// TwinCAT 3 PLC project LibraryVision
// Title: LibraryVision
// Company: Gema
// Author: RG
// ProjectVersion: 0.9.9.9
// ProgramVersion: 3.1.4024.0
// libraries:
//   Tc2_EtherCAT, * (Beckhoff Automation GmbH)
//   Tc2_System, * (Beckhoff Automation GmbH)
//   TcoCore, 0.11.0.23 (Vortex.Library)
//   TcoData, 0.11.0.23 (Vortex.Library)
//   TcoDrivesBeckhoff, 0.11.0.23 (Vortex.Library)
//   TcoElements, 0.11.0.23 (Vortex.Library)
//   TcoIo, 0.11.0.23 (Vortex.Library)
//   TcoPneumatics, 0.11.0.23 (Vortex.Library)
// project tree:
//   Context/ MainStation.TcPOU, PRG_TEST.TcPOU, TcUnitContext.TcPOU
//   IV3/Dut/CoE/ GeneralDeviceInformation.TcDUT, IdentityCoe.TcDUT
//   IV3/Dut/ Coordinates.TcDUT, FieldOfView.TcDUT
//   IV3/Dut/IO/Base/ EtcMasterBase_62654B43.TcDUT, EtcSlaveBase_82538BE2.TcDUT, EtcSlaveBoxBase_77A0E4A7.TcDUT, EtcSlaveEndTerminalBase_866C7F0C.TcDUT, EtcSlaveTerminalBase_947E5A46.TcDUT, InputBase_8311D824.TcDUT, OutputBase_10CEE7DE.TcDUT, SyncUnitsBase_AD6C35CE.TcDUT, SyncUnitTaskBase_FCD3CBF3.TcDUT, SyncUnitTasksBase_7C8711EB.TcDUT
//   IV3/Dut/IO/Devices/ SyncUnits_67D36DDA.TcDUT, SyncUnitTasks_4BE01469.TcDUT, SyncUnitTask_AB2F5079.TcDUT
//   IV3/Dut/IO/PDOs/BitValues/ Iv3InputRequestResponse1.TcDUT, Iv3InputRequestResponse2.TcDUT, Iv3InputRequestResponse3.TcDUT, Iv3InputRequestResponse4.TcDUT (not stored), Iv3InputRequestResponse5.TcDUT
//   IV3/Dut/IO/PDOs/ ID01_Current_Value.TcDUT, ID01_Status.TcDUT, ID02_Current_Value.TcDUT, ID02_Status.TcDUT, ID03_Current_Value.TcDUT, ID03_Status.TcDUT, ID04_Current_Value.TcDUT, ID04_Status.TcDUT, ID05_Current_Value.TcDUT, ID05_Status.TcDUT, ID06_Current_Value.TcDUT, ID06_Status.TcDUT, ID07_Current_Value.TcDUT, ID07_Status.TcDUT, ID08_Current_Value.TcDUT, ID08_Status.TcDUT, InfoData.TcDUT, InfoData_8649EEEB.TcDUT, InfoData_E68C61CD.TcDUT, Inputs.TcDUT, Input_Request.TcDUT, Input_Response.TcDUT, Outputs.TcDUT, Status_of_System.TcDUT, WcState_0B2B16F9.TcDUT, WcState_9091E0EB.TcDUT
//   IV3/Interfaces/ iCalculationTask.TcIO
//   IV3/ IVController.TcPOU
//   IV3/Tasks/ ReadCoordinates.TcPOU, CalculationTask.TcPOU, TriggerSensor.TcPOU
//   Project Information/ F_GetCompany.TcPOU, F_GetTitle.TcPOU, F_GetVersion.TcPOU
//   Version/ Global_Version.TcGVL
// real-time tasks:
//   TASK PlcTask: cycle T#1ms, priority 20, ADS port 350
// I/O:
//   DEVICE Device 2 (EtherCAT), AmsNetId 192.168.1.8.3.1
//     IV3_Sensor1(DL-EC1A)
// variable links:
//   LibraryVisionExample Instance <-> Device 2 (EtherCAT)/IV3_Sensor1(DL-EC1A)
//     PlcTask Inputs/MAIN._app._mainStation._IvController.ID01Status/Change_Program_Ack <-> ID01 Status/Change Program Ack
//     PlcTask Inputs/MAIN._app._mainStation._IvController.ID01Status/Change_Program_Failed <-> ID01 Status/Change Program Failed
//     PlcTask Inputs/MAIN._app._mainStation._IvController.ID01Status/Error_status <-> ID01 Status/Error status
//     PlcTask Inputs/MAIN._app._mainStation._IvController.ID01Status/Program_Num_00 <-> ID01 Status/Program Num 00
//     PlcTask Inputs/MAIN._app._mainStation._IvController.ID02Status/Program_Num_01 <-> ID02 Status/Program Num 01
//     PlcTask Inputs/MAIN._app._mainStation._IvController.ID03Status/Program_Num_02 <-> ID03 Status/Program Num 02
//     PlcTask Inputs/MAIN._app._mainStation._IvController.ID04Status/Program_Num_03 <-> ID04 Status/Program Num 03
//     PlcTask Inputs/MAIN._app._mainStation._IvController.ID05Status/Program_Num_04 <-> ID05 Status/Program Num 04
//     PlcTask Inputs/MAIN._app._mainStation._IvController.ID06Status/Program_Num_05 <-> ID06 Status/Program Num 05
//     PlcTask Inputs/MAIN._app._mainStation._IvController.ID07Status/Program_Num_06 <-> ID07 Status/Program Num 06
//     PlcTask Inputs/MAIN._app._mainStation._IvController.ID01Status/Result_Valid <-> ID01 Status/Result Valid
//     PlcTask Inputs/MAIN._app._mainStation._IvController.ID01Status/Total_Status_OK <-> ID01 Status/Total Status OK
//     PlcTask Inputs/MAIN._app._mainStation._IvController.ID03Status/Total_Status_OK <-> ID03 Status/Total Status OK
//     PlcTask Inputs/MAIN._app._mainStation._IvController.ID01_CurrentValue/Reserved <-> ID01 Current Value/Reserved
//     PlcTask Inputs/MAIN._app._mainStation._IvController.ID02Status/Result_Updated_Toggle <-> ID02 Status/Result Updated Toggle
//     PlcTask Inputs/MAIN._app._mainStation._IvController.ID02Status/Tool_00_Invalid <-> ID02 Status/Tool 00 Invalid
//     PlcTask Inputs/MAIN._app._mainStation._IvController.ID03Status/Tool_01_Invalid <-> ID03 Status/Tool 01 Invalid
//     PlcTask Inputs/MAIN._app._mainStation._IvController.ID04Status/Tool_02_Invalid <-> ID04 Status/Tool 02 Invalid
//     PlcTask Inputs/MAIN._app._mainStation._IvController.ID05Status/Tool_03_Invalid <-> ID05 Status/Tool 03 Invalid
//     PlcTask Inputs/MAIN._app._mainStation._IvController.ID06Status/Tool_04_Invalid <-> ID06 Status/Tool 04 Invalid
//     PlcTask Inputs/MAIN._app._mainStation._IvController.ID07Status/Tool_05_Invalid <-> ID07 Status/Tool 05 Invalid
//     PlcTask Inputs/MAIN._app._mainStation._IvController.ID08Status/Tool_06_Invalid <-> ID08 Status/Tool 06 Invalid
//     PlcTask Inputs/MAIN._app._mainStation._IvController.ID02Status/Tool_00_Status <-> ID02 Status/Tool 00 Status
//     PlcTask Inputs/MAIN._app._mainStation._IvController.ID03Status/Tool_01_Status <-> ID03 Status/Tool 01 Status
//     PlcTask Inputs/MAIN._app._mainStation._IvController.ID04Status/Tool_02_Status <-> ID04 Status/Tool 02 Status
//     PlcTask Inputs/MAIN._app._mainStation._IvController.ID05Status/Tool_03_Status <-> ID05 Status/Tool 03 Status
//     PlcTask Inputs/MAIN._app._mainStation._IvController.ID06Status/Tool_04_Status <-> ID06 Status/Tool 04 Status
//     PlcTask Inputs/MAIN._app._mainStation._IvController.ID07Status/Tool_05_Status <-> ID07 Status/Tool 05 Status
//     PlcTask Inputs/MAIN._app._mainStation._IvController.ID08Status/Tool_06_Status <-> ID08 Status/Tool 06 Status
//     PlcTask Inputs/MAIN._app._mainStation._IvController.ID02Status/Trigger_Ack <-> ID02 Status/Trigger Ack
//     PlcTask Inputs/MAIN._app._mainStation._IvController.ID02Status/Trigger_Failed <-> ID02 Status/Trigger Failed
//     PlcTask Inputs/MAIN._app._mainStation._IvController.ID02_MatchingRateOfPositionAdujustmentTool_01/Tool_00_Score <-> ID02 Current Value/Tool 00 Score
//     PlcTask Inputs/MAIN._app._mainStation._IvController.ID03_MatchingRateOfPositionAdujustmentTool_02/Tool_01_Score <-> ID03 Current Value/Tool 01 Score
//     PlcTask Inputs/MAIN._app._mainStation._IvController.ID04_MatchingRateOfPositionAdujustmentTool_03/Tool_02_Score <-> ID04 Current Value/Tool 02 Score
//     PlcTask Inputs/MAIN._app._mainStation._IvController.ID05_MatchingRateOfPositionAdujustmentTool_04/Tool_03_Score <-> ID05 Current Value/Tool 03 Score
//     PlcTask Inputs/MAIN._app._mainStation._IvController.ID06_MatchingRateOfPositionAdujustmentTool_05/Tool_04_Score <-> ID06 Current Value/Tool 04 Score
//     PlcTask Inputs/MAIN._app._mainStation._IvController.ID07_MatchingRateOfPositionAdujustmentTool_06/Tool_05_Score <-> ID07 Current Value/Tool 05 Score
//     PlcTask Inputs/MAIN._app._mainStation._IvController.ID08_MatchingRateOfPositionAdujustmentTool_07/Tool_06_Score <-> ID08 Current Value/Tool 06 Score
//     PlcTask Inputs/MAIN._app._mainStation._IvController.ID03Status/Regist_Master_Image_Ack <-> ID03 Status/Regist Master Image Ack
//     PlcTask Inputs/MAIN._app._mainStation._IvController.ID03Status/Regist_Master_Image_Failed <-> ID03 Status/Regist Master Image Failed
//     PlcTask Inputs/MAIN._app._mainStation._IvController.ID04Status/Logic_01 <-> ID04 Status/Logic 01
//     PlcTask Inputs/MAIN._app._mainStation._IvController.ID05Status/Logic_02 <-> ID05 Status/Logic 02
//     PlcTask Inputs/MAIN._app._mainStation._IvController.ID06Status/Logic_03 <-> ID06 Status/Logic 03
//     PlcTask Inputs/MAIN._app._mainStation._IvController.ID07Status/Logic_04 <-> ID07 Status/Logic 04
//     PlcTask Inputs/MAIN._app._mainStation._IvController.ID04Status/SD_Card_Detected <-> ID04 Status/SD Card Detected
//     PlcTask Inputs/MAIN._app._mainStation._IvController.ID04Status/SD_Save_Stop_Ack <-> ID04 Status/SD Save Stop Ack
//     PlcTask Inputs/MAIN._app._mainStation._IvController.ID05Status/Reset_Statistics_Ack <-> ID05 Status/Reset Statistics Ack
//     PlcTask Inputs/MAIN._app._mainStation._IvController.ID05Status/Run <-> ID05 Status/Run
//     PlcTask Inputs/MAIN._app._mainStation._IvController.ID06Status/Busy <-> ID06 Status/Busy
//     PlcTask Inputs/MAIN._app._mainStation._IvController.ID06Status/Clear_Error_Ack <-> ID06 Status/Clear Error Ack
//     PlcTask Inputs/MAIN._app._mainStation._IvController.ID08Status/SD_Card_No_Space <-> ID08 Status/SD Card No Space
//     PlcTask Inputs/MAIN._app._mainStation._IvController.ID08Status/Total_Status_NG <-> ID08 Status/Total Status NG
//     PlcTask Inputs/MAIN._app._mainStation._IvController.InfoData/AdsAddr <-> InfoData/AdsAddr
//     PlcTask Inputs/MAIN._app._mainStation._IvController.InfoData/State <-> InfoData/State
//     PlcTask Inputs/MAIN._app._mainStation._IvController.InputResponse/Response_{1..5} <-> Input Response {1..5}/Reserved  (5 links)
//     PlcTask Inputs/MAIN._app._mainStation._IvController.StatusOfSystem/Error_Code <-> Status of System/Error Code
//     PlcTask Inputs/MAIN._app._mainStation._IvController.StatusOfSystem/Error_Status <-> Status of System/Error Status
//     PlcTask Inputs/MAIN._app._mainStation._IvController.WcState/WcState <-> WcState/WcState
//     PlcTask Outputs/MAIN._app._mainStation._IvController.InputRequest/Request_{1..5} <-> Input Request {1..5}/Request {1..5}  (5 links)

// ---- IV3/Dut/CoE/GeneralDeviceInformation.TcDUT
TYPE
    GeneralDeviceInformation :
    STRUCT
        DeviceType      : UDINT;
        DeviceName      : STRING;
        HardwareVersion : STRING;
        SoftwareVersion : STRING;
    END_STRUCT
END_TYPE

// ---- IV3/Dut/CoE/IdentityCoe.TcDUT
TYPE
    IdentityCoe :
    STRUCT
        VendorId     : DWORD;
        ProductKey   : DWORD;
        Revision     : DWORD;
        SerialNumber : DWORD;
    END_STRUCT
END_TYPE

// ---- IV3/Dut/Coordinates.TcDUT
TYPE
    Coordinates :
    STRUCT
        xValue        : DINT;
        yValue        : DINT;
        variableValue : DINT;
    END_STRUCT
END_TYPE

// ---- IV3/Dut/FieldOfView.TcDUT
TYPE
    FieldOfView :
    STRUCT
        xValue : LREAL;
        yValue : lreal;
    END_STRUCT
END_TYPE

// ---- IV3/Dut/IO/Base/EtcMasterBase_62654B43.TcDUT

TYPE
    EtcMasterBase_62654B43 :
    STRUCT
    END_STRUCT
END_TYPE

// ---- IV3/Dut/IO/Base/EtcSlaveBase_82538BE2.TcDUT

TYPE
    EtcSlaveBase_82538BE2 :
    STRUCT
    END_STRUCT
END_TYPE

// ---- IV3/Dut/IO/Base/EtcSlaveBoxBase_77A0E4A7.TcDUT

{attribute clr[Container(Layout.Stack)]}
{attribute clr[Group(Layout.GroupBox)]}
{attribute addProperty PreviousPort "Unknown"}
{attribute addProperty SyncUnit "Unknown"}
TYPE
    EtcSlaveBoxBase_77A0E4A7 EXTENDS EtcSlaveBase_82538BE2 :
    STRUCT
    END_STRUCT
END_TYPE

// ---- IV3/Dut/IO/Base/EtcSlaveEndTerminalBase_866C7F0C.TcDUT

{attribute clr[Container(Layout.Stack)]}
{attribute clr[Group(Layout.GroupBox)]}
{attribute addProperty PreviousPort "Unknown"}
{attribute addProperty SyncUnit "Unknown"}
TYPE
    EtcSlaveEndTerminalBase_866C7F0C EXTENDS EtcSlaveBase_82538BE2 :
    STRUCT
    END_STRUCT
END_TYPE

// ---- IV3/Dut/IO/Base/EtcSlaveTerminalBase_947E5A46.TcDUT

{attribute clr[Container(Layout.Stack)]}
{attribute clr[Group(Layout.GroupBox)]}
{attribute addProperty PreviousPort "Unknown"}
{attribute addProperty SyncUnit "Unknown"}
TYPE
    EtcSlaveTerminalBase_947E5A46 EXTENDS EtcSlaveBase_82538BE2 :
    STRUCT
    END_STRUCT
END_TYPE

// ---- IV3/Dut/IO/Base/InputBase_8311D824.TcDUT

TYPE
    InputBase_8311D824 :
    STRUCT
    END_STRUCT
END_TYPE

// ---- IV3/Dut/IO/Base/OutputBase_10CEE7DE.TcDUT

TYPE
    OutputBase_10CEE7DE :
    STRUCT
    END_STRUCT
END_TYPE

// ---- IV3/Dut/IO/Base/SyncUnitsBase_AD6C35CE.TcDUT

TYPE
    SyncUnitsBase_AD6C35CE :
    STRUCT
    END_STRUCT
END_TYPE

// ---- IV3/Dut/IO/Base/SyncUnitTaskBase_FCD3CBF3.TcDUT

TYPE
    SyncUnitTaskBase_FCD3CBF3 :
    STRUCT
    END_STRUCT
END_TYPE

// ---- IV3/Dut/IO/Base/SyncUnitTasksBase_7C8711EB.TcDUT

TYPE
    SyncUnitTasksBase_7C8711EB :
    STRUCT
    END_STRUCT
END_TYPE

// ---- IV3/Dut/IO/Devices/SyncUnits_67D36DDA.TcDUT
{attribute 'GeneratedUsingTerminal: '}
{attribute addProperty BoxType ""}
{attribute addProperty Id "_defaultAT %I*SyncUnitTasks_4BE0146918"}
{attribute addProperty CRC "1741909466"}
{attribute addProperty Size "18"}
TYPE
    SyncUnits_67D36DDA EXTENDS SyncUnitsBase_AD6C35CE :
    STRUCT
        {attribute addProperty Name "_default"}
        _default : SyncUnitTasks_4BE01469;
    END_STRUCT
END_TYPE

// ---- IV3/Dut/IO/Devices/SyncUnitTasks_4BE01469.TcDUT
{attribute 'GeneratedUsingTerminal: '}
{attribute addProperty BoxType ""}
{attribute addProperty Id "unreferencedAT %I*SyncUnitTask_AB2F50799PlcTaskAT %I*SyncUnitTask_AB2F50799"}
{attribute addProperty CRC "1272976489"}
{attribute addProperty Size "18"}
TYPE
    SyncUnitTasks_4BE01469 EXTENDS SyncUnitTasksBase_7C8711EB :
    STRUCT
        {attribute addProperty Name "unreferenced"}
        unreferenced : SyncUnitTask_AB2F5079;
        {attribute addProperty Name "PlcTask"}
        PlcTask : SyncUnitTask_AB2F5079;
    END_STRUCT
END_TYPE

// ---- IV3/Dut/IO/Devices/SyncUnitTask_AB2F5079.TcDUT
{attribute 'GeneratedUsingTerminal: IODEVICETYPE_ETHERCATPROT'}
{attribute addProperty BoxType "IODEVICETYPE_ETHERCATPROT"}
{attribute addProperty Id "WcStateAT %I*WcState_0B2B16F91InfoDataAT %I*InfoData_8649EEEB8"}
{attribute addProperty CRC "2872004729"}
{attribute addProperty Size "9"}
TYPE
    SyncUnitTask_AB2F5079 EXTENDS SyncUnitTaskBase_FCD3CBF3 :
    STRUCT
        {attribute addProperty Name "WcState"}
        WcState : WcState_0B2B16F9;
        {attribute addProperty Name "InfoData"}
        InfoData : InfoData_8649EEEB;
    END_STRUCT
END_TYPE

// ---- IV3/Dut/IO/PDOs/BitValues/Iv3InputRequestResponse1.TcDUT
//Index0x7000   Subindex 16#1
TYPE
    Iv3InputRequestResponse1 :
    STRUCT
        Bit0                      : BIT;
        ProgramChangeRequest      : BIT;
        Trigger                   : BIT;
        MasterRegistrationRequest : BIT;
        MemoryStopSdCardRequest   : BIT;
        ResetStatistics           : BIT;
        ResetError                : BIT;
        Bit7                      : BIT;
        Bit8                      : BIT;
        Bit9                      : BIT;
        Bit10                     : BIT;
        Bit11                     : BIT;
        Bit12                     : BIT;
        Bit13                     : BIT;
        Bit14                     : BIT;
        Bit15                     : BIT;

    END_STRUCT
END_TYPE

// ---- IV3/Dut/IO/PDOs/BitValues/Iv3InputRequestResponse2.TcDUT
//Index0x7000   Subindex 16#2
TYPE
    Iv3InputRequestResponse2 :
    STRUCT
        Bit0                     : BIT;
        SwitchProgrammNumberBit0 : BIT;
        Bit2                     : BIT;
        Bit3                     : BIT;
        Bit4                     : BIT;
        Bit5                     : BIT;
        Bit6                     : BIT;
        Bit7                     : BIT;
        Bit8                     : BIT;
        Bit9                     : BIT;
        Bit10                    : BIT;
        Bit11                    : BIT;
        Bit12                    : BIT;
        Bit13                    : BIT;
        Bit14                    : BIT;
        Bit15                    : BIT;

    END_STRUCT
END_TYPE

// ---- IV3/Dut/IO/PDOs/BitValues/Iv3InputRequestResponse3.TcDUT
//Index0x7000   Subindex 16#3
TYPE
    Iv3InputRequestResponse3 :
    STRUCT
        Bit0                     : BIT;
        SwitchProgrammNumberBit1 : BIT;
        Bit2                     : BIT;
        Bit3                     : BIT;
        Bit4                     : BIT;
        Bit5                     : BIT;
        Bit6                     : BIT;
        Bit7                     : BIT;
        Bit8                     : BIT;
        Bit9                     : BIT;
        Bit10                    : BIT;
        Bit11                    : BIT;
        Bit12                    : BIT;
        Bit13                    : BIT;
        Bit14                    : BIT;
        Bit15                    : BIT;

    END_STRUCT
END_TYPE

// ---- IV3/Dut/IO/PDOs/BitValues/Iv3InputRequestResponse5.TcDUT
//Index0x7000   Subindex 16#5
TYPE
    Iv3InputRequestResponse5 :
    STRUCT
        Bit0                     : BIT;
        SwitchProgrammNumberBit3 : BIT;
        Bit2                     : BIT;
        Bit3                     : BIT;
        Bit4                     : BIT;
        Bit5                     : BIT;
        Bit6                     : BIT;
        Bit7                     : BIT;
        Bit8                     : BIT;
        Bit9                     : BIT;
        Bit10                    : BIT;
        Bit11                    : BIT;
        Bit12                    : BIT;
        Bit13                    : BIT;
        Bit14                    : BIT;
        Bit15                    : BIT;

    END_STRUCT
END_TYPE

// ---- IV3/Dut/IO/PDOs/ID01_Current_Value.TcDUT
{attribute 'GeneratedUsingTerminal: DL-EC1A-0000'}
{attribute addProperty BoxType "DL-EC1A-0000"}
{attribute addProperty Id "ReservedAT %I*DINT4"}
{attribute addProperty CRC "2013026300"}
{attribute addProperty Size "4"}
TYPE
    ID01_Current_Value EXTENDS InputBase_8311D824 :
    STRUCT
        {attribute addProperty Name "Reserved"}
        Reserved AT %I* : DINT;
    END_STRUCT
END_TYPE

// ---- IV3/Dut/IO/PDOs/ID01_Status.TcDUT
{attribute 'GeneratedUsingTerminal: DL-EC1A-0000'}
{attribute addProperty BoxType "DL-EC1A-0000"}
{attribute addProperty Id "Change_Program_AckAT %I*BOOL1Change_Program_FailedAT %I*BOOL1Result_ValidAT %I*BOOL1Total_Status_OKAT %I*BOOL1Program_Num_00AT %I*BOOL1Error_statusAT %I*BOOL1"}
{attribute addProperty CRC "3787914147"}
{attribute addProperty Size "6"}
TYPE
    ID01_Status EXTENDS InputBase_8311D824 :
    STRUCT
        {attribute addProperty Name "Change_Program_Ack"}
        Change_Program_Ack AT %I* : BOOL;
        {attribute addProperty Name "Change_Program_Failed"}
        Change_Program_Failed AT %I* : BOOL;
        {attribute addProperty Name "Result_Valid"}
        Result_Valid AT %I* : BOOL;
        {attribute addProperty Name "Total_Status_OK"}
        Total_Status_OK AT %I* : BOOL;
        {attribute addProperty Name "Program_Num_00"}
        Program_Num_00 AT %I* : BOOL;
        {attribute addProperty Name "Error_status"}
        Error_status AT %I* : BOOL;
    END_STRUCT
END_TYPE

// ---- IV3/Dut/IO/PDOs/ID02_Current_Value.TcDUT
{attribute 'GeneratedUsingTerminal: DL-EC1A-0000'}
{attribute addProperty BoxType "DL-EC1A-0000"}
{attribute addProperty Id "Tool_00_ScoreAT %I*DINT4"}
{attribute addProperty CRC "539608926"}
{attribute addProperty Size "4"}
TYPE
    ID02_Current_Value EXTENDS InputBase_8311D824 :
    STRUCT
        {attribute addProperty Name "Tool_00_Score"}
        Tool_00_Score AT %I* : DINT;
    END_STRUCT
END_TYPE

// ---- IV3/Dut/IO/PDOs/ID02_Status.TcDUT
{attribute 'GeneratedUsingTerminal: DL-EC1A-0000'}
{attribute addProperty BoxType "DL-EC1A-0000"}
{attribute addProperty Id "Trigger_AckAT %I*BOOL1Trigger_FailedAT %I*BOOL1Result_Updated_ToggleAT %I*BOOL1Tool_00_StatusAT %I*BOOL1Program_Num_01AT %I*BOOL1Tool_00_InvalidAT %I*BOOL1"}
{attribute addProperty CRC "3351424392"}
{attribute addProperty Size "6"}
TYPE
    ID02_Status EXTENDS InputBase_8311D824 :
    STRUCT
        {attribute addProperty Name "Trigger_Ack"}
        Trigger_Ack AT %I* : BOOL;
        {attribute addProperty Name "Trigger_Failed"}
        Trigger_Failed AT %I* : BOOL;
        {attribute addProperty Name "Result_Updated_Toggle"}
        Result_Updated_Toggle AT %I* : BOOL;
        {attribute addProperty Name "Tool_00_Status"}
        Tool_00_Status AT %I* : BOOL;
        {attribute addProperty Name "Program_Num_01"}
        Program_Num_01 AT %I* : BOOL;
        {attribute addProperty Name "Tool_00_Invalid"}
        Tool_00_Invalid AT %I* : BOOL;
    END_STRUCT
END_TYPE

// ---- IV3/Dut/IO/PDOs/ID03_Current_Value.TcDUT
{attribute 'GeneratedUsingTerminal: DL-EC1A-0000'}
{attribute addProperty BoxType "DL-EC1A-0000"}
{attribute addProperty Id "Tool_01_ScoreAT %I*DINT4"}
{attribute addProperty CRC "2706247979"}
{attribute addProperty Size "4"}
TYPE
    ID03_Current_Value EXTENDS InputBase_8311D824 :
    STRUCT
        {attribute addProperty Name "Tool_01_Score"}
        Tool_01_Score AT %I* : DINT;
    END_STRUCT
END_TYPE

// ---- IV3/Dut/IO/PDOs/ID03_Status.TcDUT
{attribute 'GeneratedUsingTerminal: DL-EC1A-0000'}
{attribute addProperty BoxType "DL-EC1A-0000"}
{attribute addProperty Id "Regist_Master_Image_AckAT %I*BOOL1Regist_Master_Image_FailedAT %I*BOOL1Total_Status_OKAT %I*BOOL1Tool_01_StatusAT %I*BOOL1Program_Num_02AT %I*BOOL1Tool_01_InvalidAT %I*BOOL1"}
{attribute addProperty CRC "695297954"}
{attribute addProperty Size "6"}
TYPE
    ID03_Status EXTENDS InputBase_8311D824 :
    STRUCT
        {attribute addProperty Name "Regist_Master_Image_Ack"}
        Regist_Master_Image_Ack AT %I* : BOOL;
        {attribute addProperty Name "Regist_Master_Image_Failed"}
        Regist_Master_Image_Failed AT %I* : BOOL;
        {attribute addProperty Name "Total_Status_OK"}
        Total_Status_OK AT %I* : BOOL;
        {attribute addProperty Name "Tool_01_Status"}
        Tool_01_Status AT %I* : BOOL;
        {attribute addProperty Name "Program_Num_02"}
        Program_Num_02 AT %I* : BOOL;
        {attribute addProperty Name "Tool_01_Invalid"}
        Tool_01_Invalid AT %I* : BOOL;
    END_STRUCT
END_TYPE

// ---- IV3/Dut/IO/PDOs/ID04_Current_Value.TcDUT
{attribute 'GeneratedUsingTerminal: DL-EC1A-0000'}
{attribute addProperty BoxType "DL-EC1A-0000"}
{attribute addProperty Id "Tool_02_ScoreAT %I*DINT4"}
{attribute addProperty CRC "640120323"}
{attribute addProperty Size "4"}
TYPE
    ID04_Current_Value EXTENDS InputBase_8311D824 :
    STRUCT
        {attribute addProperty Name "Tool_02_Score"}
        Tool_02_Score AT %I* : DINT;
    END_STRUCT
END_TYPE

// ---- IV3/Dut/IO/PDOs/ID04_Status.TcDUT
{attribute 'GeneratedUsingTerminal: DL-EC1A-0000'}
{attribute addProperty BoxType "DL-EC1A-0000"}
{attribute addProperty Id "SD_Save_Stop_AckAT %I*BOOL1SD_Card_DetectedAT %I*BOOL1Logic_01AT %I*BOOL1Tool_02_StatusAT %I*BOOL1Program_Num_03AT %I*BOOL1Tool_02_InvalidAT %I*BOOL1"}
{attribute addProperty CRC "922163961"}
{attribute addProperty Size "6"}
TYPE
    ID04_Status EXTENDS InputBase_8311D824 :
    STRUCT
        {attribute addProperty Name "SD_Save_Stop_Ack"}
        SD_Save_Stop_Ack AT %I* : BOOL;
        {attribute addProperty Name "SD_Card_Detected"}
        SD_Card_Detected AT %I* : BOOL;
        {attribute addProperty Name "Logic_01"}
        Logic_01 AT %I* : BOOL;
        {attribute addProperty Name "Tool_02_Status"}
        Tool_02_Status AT %I* : BOOL;
        {attribute addProperty Name "Program_Num_03"}
        Program_Num_03 AT %I* : BOOL;
        {attribute addProperty Name "Tool_02_Invalid"}
        Tool_02_Invalid AT %I* : BOOL;
    END_STRUCT
END_TYPE

// ---- IV3/Dut/IO/PDOs/ID05_Current_Value.TcDUT
{attribute 'GeneratedUsingTerminal: DL-EC1A-0000'}
{attribute addProperty BoxType "DL-EC1A-0000"}
{attribute addProperty Id "Tool_03_ScoreAT %I*DINT4"}
{attribute addProperty CRC "2806030454"}
{attribute addProperty Size "4"}
TYPE
    ID05_Current_Value EXTENDS InputBase_8311D824 :
    STRUCT
        {attribute addProperty Name "Tool_03_Score"}
        Tool_03_Score AT %I* : DINT;
    END_STRUCT
END_TYPE

// ---- IV3/Dut/IO/PDOs/ID05_Status.TcDUT
{attribute 'GeneratedUsingTerminal: DL-EC1A-0000'}
{attribute addProperty BoxType "DL-EC1A-0000"}
{attribute addProperty Id "Reset_Statistics_AckAT %I*BOOL1RunAT %I*BOOL1Logic_02AT %I*BOOL1Tool_03_StatusAT %I*BOOL1Program_Num_04AT %I*BOOL1Tool_03_InvalidAT %I*BOOL1"}
{attribute addProperty CRC "2929837159"}
{attribute addProperty Size "6"}
TYPE
    ID05_Status EXTENDS InputBase_8311D824 :
    STRUCT
        {attribute addProperty Name "Reset_Statistics_Ack"}
        Reset_Statistics_Ack AT %I* : BOOL;
        {attribute addProperty Name "Run"}
        Run AT %I* : BOOL;
        {attribute addProperty Name "Logic_02"}
        Logic_02 AT %I* : BOOL;
        {attribute addProperty Name "Tool_03_Status"}
        Tool_03_Status AT %I* : BOOL;
        {attribute addProperty Name "Program_Num_04"}
        Program_Num_04 AT %I* : BOOL;
        {attribute addProperty Name "Tool_03_Invalid"}
        Tool_03_Invalid AT %I* : BOOL;
    END_STRUCT
END_TYPE

// ---- IV3/Dut/IO/PDOs/ID06_Current_Value.TcDUT
{attribute 'GeneratedUsingTerminal: DL-EC1A-0000'}
{attribute addProperty BoxType "DL-EC1A-0000"}
{attribute addProperty Id "Tool_04_ScoreAT %I*DINT4"}
{attribute addProperty CRC "741647844"}
{attribute addProperty Size "4"}
TYPE
    ID06_Current_Value EXTENDS InputBase_8311D824 :
    STRUCT
        {attribute addProperty Name "Tool_04_Score"}
        Tool_04_Score AT %I* : DINT;
    END_STRUCT
END_TYPE

// ---- IV3/Dut/IO/PDOs/ID06_Status.TcDUT
{attribute 'GeneratedUsingTerminal: DL-EC1A-0000'}
{attribute addProperty BoxType "DL-EC1A-0000"}
{attribute addProperty Id "Clear_Error_AckAT %I*BOOL1BusyAT %I*BOOL1Logic_03AT %I*BOOL1Tool_04_StatusAT %I*BOOL1Program_Num_05AT %I*BOOL1Tool_04_InvalidAT %I*BOOL1"}
{attribute addProperty CRC "1399145824"}
{attribute addProperty Size "6"}
TYPE
    ID06_Status EXTENDS InputBase_8311D824 :
    STRUCT
        {attribute addProperty Name "Clear_Error_Ack"}
        Clear_Error_Ack AT %I* : BOOL;
        {attribute addProperty Name "Busy"}
        Busy AT %I* : BOOL;
        {attribute addProperty Name "Logic_03"}
        Logic_03 AT %I* : BOOL;
        {attribute addProperty Name "Tool_04_Status"}
        Tool_04_Status AT %I* : BOOL;
        {attribute addProperty Name "Program_Num_05"}
        Program_Num_05 AT %I* : BOOL;
        {attribute addProperty Name "Tool_04_Invalid"}
        Tool_04_Invalid AT %I* : BOOL;
    END_STRUCT
END_TYPE

// ---- IV3/Dut/IO/PDOs/ID07_Current_Value.TcDUT
{attribute 'GeneratedUsingTerminal: DL-EC1A-0000'}
{attribute addProperty BoxType "DL-EC1A-0000"}
{attribute addProperty Id "Tool_05_ScoreAT %I*DINT4"}
{attribute addProperty CRC "2907927441"}
{attribute addProperty Size "4"}
TYPE
    ID07_Current_Value EXTENDS InputBase_8311D824 :
    STRUCT
        {attribute addProperty Name "Tool_05_Score"}
        Tool_05_Score AT %I* : DINT;
    END_STRUCT
END_TYPE

// ---- IV3/Dut/IO/PDOs/ID07_Status.TcDUT
{attribute 'GeneratedUsingTerminal: DL-EC1A-0000'}
{attribute addProperty BoxType "DL-EC1A-0000"}
{attribute addProperty Id "Logic_04AT %I*BOOL1Tool_05_StatusAT %I*BOOL1Program_Num_06AT %I*BOOL1Tool_05_InvalidAT %I*BOOL1"}
{attribute addProperty CRC "1568950313"}
{attribute addProperty Size "4"}
TYPE
    ID07_Status EXTENDS InputBase_8311D824 :
    STRUCT
        {attribute addProperty Name "Logic_04"}
        Logic_04 AT %I* : BOOL;
        {attribute addProperty Name "Tool_05_Status"}
        Tool_05_Status AT %I* : BOOL;
        {attribute addProperty Name "Program_Num_06"}
        Program_Num_06 AT %I* : BOOL;
        {attribute addProperty Name "Tool_05_Invalid"}
        Tool_05_Invalid AT %I* : BOOL;
    END_STRUCT
END_TYPE

// ---- IV3/Dut/IO/PDOs/ID08_Current_Value.TcDUT
{attribute 'GeneratedUsingTerminal: DL-EC1A-0000'}
{attribute addProperty BoxType "DL-EC1A-0000"}
{attribute addProperty Id "Tool_06_ScoreAT %I*DINT4"}
{attribute addProperty CRC "708449465"}
{attribute addProperty Size "4"}
TYPE
    ID08_Current_Value EXTENDS InputBase_8311D824 :
    STRUCT
        {attribute addProperty Name "Tool_06_Score"}
        Tool_06_Score AT %I* : DINT;
    END_STRUCT
END_TYPE

// ---- IV3/Dut/IO/PDOs/ID08_Status.TcDUT
{attribute 'GeneratedUsingTerminal: DL-EC1A-0000'}
{attribute addProperty BoxType "DL-EC1A-0000"}
{attribute addProperty Id "SD_Card_No_SpaceAT %I*BOOL1Total_Status_NGAT %I*BOOL1Tool_06_StatusAT %I*BOOL1Tool_06_InvalidAT %I*BOOL1"}
{attribute addProperty CRC "795074029"}
{attribute addProperty Size "4"}
TYPE
    ID08_Status EXTENDS InputBase_8311D824 :
    STRUCT
        {attribute addProperty Name "SD_Card_No_Space"}
        SD_Card_No_Space AT %I* : BOOL;
        {attribute addProperty Name "Total_Status_NG"}
        Total_Status_NG AT %I* : BOOL;
        {attribute addProperty Name "Tool_06_Status"}
        Tool_06_Status AT %I* : BOOL;
        {attribute addProperty Name "Tool_06_Invalid"}
        Tool_06_Invalid AT %I* : BOOL;
    END_STRUCT
END_TYPE

// ---- IV3/Dut/IO/PDOs/InfoData.TcDUT
{attribute 'GeneratedUsingTerminal: DL-EC1A-0000'}
{attribute addProperty BoxType "DL-EC1A-0000"}
{attribute addProperty Id "AdsAddrAT %I*AMSADDR8StateAT %I*UINT2"}
{attribute addProperty CRC "854291690"}
{attribute addProperty Size "10"}
TYPE
    InfoData EXTENDS InputBase_8311D824 :
    STRUCT
        {attribute addProperty Name "AdsAddr"}
        AdsAddr AT %I* : AMSADDR;
        {attribute addProperty Name "State"}
        State AT %I* : UINT;
    END_STRUCT
END_TYPE

// ---- IV3/Dut/IO/PDOs/InfoData_8649EEEB.TcDUT
{attribute 'GeneratedUsingTerminal: IODEVICETYPE_ETHERCATPROT'}
{attribute addProperty BoxType "IODEVICETYPE_ETHERCATPROT"}
{attribute addProperty Id "ObjectIdAT %I*DWORD4StateAT %I*UINT2SlaveCountAT %I*UINT2"}
{attribute addProperty CRC "2252992235"}
{attribute addProperty Size "8"}
TYPE
    InfoData_8649EEEB EXTENDS InputBase_8311D824 :
    STRUCT
        {attribute addProperty Name "ObjectId"}
        ObjectId AT %I* : DWORD;
        {attribute addProperty Name "State"}
        State AT %I* : UINT;
        {attribute addProperty Name "SlaveCount"}
        SlaveCount AT %I* : UINT;
    END_STRUCT
END_TYPE

// ---- IV3/Dut/IO/PDOs/InfoData_E68C61CD.TcDUT
{attribute 'GeneratedUsingTerminal: IODEVICETYPE_ETHERCATPROT'}
{attribute addProperty BoxType "IODEVICETYPE_ETHERCATPROT"}
{attribute addProperty Id "ChangeCountAT %I*UINT2DevIdAT %I*UINT2AmsNetIdAT %I*AMSNETID6CfgSlaveCountAT %I*UINT2DcToTcTimeOffsetAT %I*LINT8DcToExtTimeOffsetAT %I*LINT8"}
{attribute addProperty CRC "3867959757"}
{attribute addProperty Size "28"}
TYPE
    InfoData_E68C61CD EXTENDS InputBase_8311D824 :
    STRUCT
        {attribute addProperty Name "ChangeCount"}
        ChangeCount AT %I* : UINT;
        {attribute addProperty Name "DevId"}
        DevId AT %I* : UINT;
        {attribute addProperty Name "AmsNetId"}
        AmsNetId AT %I* : AMSNETID;
        {attribute addProperty Name "CfgSlaveCount"}
        CfgSlaveCount AT %I* : UINT;
        {attribute addProperty Name "DcToTcTimeOffset"}
        DcToTcTimeOffset AT %I* : LINT;
        {attribute addProperty Name "DcToExtTimeOffset"}
        DcToExtTimeOffset AT %I* : LINT;
    END_STRUCT
END_TYPE

// ---- IV3/Dut/IO/PDOs/Inputs.TcDUT
{attribute 'GeneratedUsingTerminal: IODEVICETYPE_ETHERCATPROT'}
{attribute addProperty BoxType "IODEVICETYPE_ETHERCATPROT"}
{attribute addProperty Id "SlaveCountAT %I*UINT2DevStateAT %I*UINT2Frm0StateAT %I*UINT2Frm0WcStateAT %I*UINT2Frm0InputToggleAT %I*UINT2"}
{attribute addProperty CRC "2791287972"}
{attribute addProperty Size "10"}
TYPE
    Inputs EXTENDS InputBase_8311D824 :
    STRUCT
        {attribute addProperty Name "SlaveCount"}
        SlaveCount AT %I* : UINT;
        {attribute addProperty Name "DevState"}
        DevState AT %I* : UINT;
        {attribute addProperty Name "Frm0State"}
        Frm0State AT %I* : UINT;
        {attribute addProperty Name "Frm0WcState"}
        Frm0WcState AT %I* : UINT;
        {attribute addProperty Name "Frm0InputToggle"}
        Frm0InputToggle AT %I* : UINT;
    END_STRUCT
END_TYPE

// ---- IV3/Dut/IO/PDOs/Input_Request.TcDUT
{attribute 'GeneratedUsingTerminal: DL-EC1A-0000'}
{attribute addProperty BoxType "DL-EC1A-0000"}
{attribute addProperty Id "Request_2AT %Q*DWORD4"}
{attribute addProperty CRC "12311493"}
{attribute addProperty Size "4"}
TYPE
    Input_Request EXTENDS OutputBase_10CEE7DE :
    STRUCT
        {attribute addProperty Name "Request_1"}
        Request_1 AT %Q* : Iv3InputRequestResponse1;
        {attribute addProperty Name "Request_2"}
        Request_2 AT %Q* : Iv3InputRequestResponse2;
        {attribute addProperty Name "Request_3"}
        Request_3 AT %Q* : Iv3InputRequestResponse3;
        {attribute addProperty Name "Request_4"}
        Request_4 AT %Q* : Iv3InputRequestResponse4;
        {attribute addProperty Name "Request_5"}
        Request_5 AT %Q* : Iv3InputRequestResponse5;
    END_STRUCT
END_TYPE

// ---- IV3/Dut/IO/PDOs/Input_Response.TcDUT
{attribute 'GeneratedUsingTerminal: DL-EC1A-0000'}
{attribute addProperty BoxType "DL-EC1A-0000"}
{attribute addProperty Id "ReservedAT %I*DWORD4"}
{attribute addProperty CRC "474832865"}
{attribute addProperty Size "4"}
TYPE
    Input_Response EXTENDS InputBase_8311D824 :
    STRUCT
        {attribute addProperty Name "Response 1"}
        Response_1 AT %Q* : Iv3InputRequestResponse1;
        {attribute addProperty Name "Response 2"}
        Response_2 AT %Q* : Iv3InputRequestResponse2;
        {attribute addProperty Name "Response 3"}
        Response_3 AT %Q* : Iv3InputRequestResponse3;
        {attribute addProperty Name "Response 4"}
        Response_4 AT %Q* : Iv3InputRequestResponse4;
        {attribute addProperty Name "Response 5"}
        Response_5 AT %Q* : Iv3InputRequestResponse5;

    END_STRUCT
END_TYPE

// ---- IV3/Dut/IO/PDOs/Outputs.TcDUT
{attribute 'GeneratedUsingTerminal: IODEVICETYPE_ETHERCATPROT'}
{attribute addProperty BoxType "IODEVICETYPE_ETHERCATPROT"}
{attribute addProperty Id "DevCtrlAT %Q*UINT2Frm0CtrlAT %Q*UINT2Frm0WcCtrlAT %Q*UINT2"}
{attribute addProperty CRC "599846173"}
{attribute addProperty Size "6"}
TYPE
    Outputs EXTENDS OutputBase_10CEE7DE :
    STRUCT
        {attribute addProperty Name "DevCtrl"}
        DevCtrl AT %Q* : UINT;
        {attribute addProperty Name "Frm0Ctrl"}
        Frm0Ctrl AT %Q* : UINT;
        {attribute addProperty Name "Frm0WcCtrl"}
        Frm0WcCtrl AT %Q* : UINT;
    END_STRUCT
END_TYPE

// ---- IV3/Dut/IO/PDOs/Status_of_System.TcDUT
{attribute 'GeneratedUsingTerminal: DL-EC1A-0000'}
{attribute addProperty BoxType "DL-EC1A-0000"}
{attribute addProperty Id "Error_StatusAT %I*BOOL1Error_CodeAT %I*UINT2"}
{attribute addProperty CRC "3460174704"}
{attribute addProperty Size "3"}
TYPE
    Status_of_System EXTENDS InputBase_8311D824 :
    STRUCT
        {attribute addProperty Name "Error_Status"}
        Error_Status AT %I* : BOOL;
        {attribute addProperty Name "Error_Code"}
        Error_Code AT %I* : UINT;
    END_STRUCT
END_TYPE

// ---- IV3/Dut/IO/PDOs/WcState_0B2B16F9.TcDUT
{attribute 'GeneratedUsingTerminal: IODEVICETYPE_ETHERCATPROT'}
{attribute addProperty BoxType "IODEVICETYPE_ETHERCATPROT"}
{attribute addProperty Id "WcStateAT %I*BOOL1"}
{attribute addProperty CRC "187373305"}
{attribute addProperty Size "1"}
TYPE
    WcState_0B2B16F9 :
    STRUCT
        {attribute addProperty Name "WcState"}
        WcState AT %I* : BOOL;
    END_STRUCT
END_TYPE

// ---- IV3/Dut/IO/PDOs/WcState_9091E0EB.TcDUT
{attribute 'GeneratedUsingTerminal: DL-EC1A-0000'}
{attribute addProperty BoxType "DL-EC1A-0000"}
{attribute addProperty Id "WcStateAT %I*BOOL1InputToggleAT %I*BOOL1"}
{attribute addProperty CRC "2425479403"}
{attribute addProperty Size "2"}
TYPE
    WcState_9091E0EB :
    STRUCT
        {attribute addProperty Name "WcState"}
        WcState AT %I* : BOOL;
        {attribute addProperty Name "InputToggle"}
        InputToggle AT %I* : BOOL;
    END_STRUCT
END_TYPE

// ---- Version/Global_Version.TcGVL
{attribute 'TcGenerated'}
{attribute 'no-analysis'}
{attribute 'linkalways'}
// This function has been automatically generated from the project information.
VAR_GLOBAL CONSTANT
    {attribute 'const_non_replaced'}
    stLibVersion_LibraryVision : ST_LibVersion :=
    (
        iMajor      := 0
        , iMinor    := 9
        , iBuild    := 9
        , iRevision := 9
        , nFlags    := 0
        , sVersion  := '0.9.9.9'
    );
END_VAR

// ---- IV3/Interfaces/iCalculationTask.TcIO
INTERFACE iCalculationTask EXTENDS TcoCore.ITcoTask

PROPERTY CoordinatesInMillimeter : REFERENCE TO Coordinates
GET
END_GET
END_PROPERTY

PROPERTY DistanceFromObject : LREAL
GET
END_GET
END_PROPERTY

PROPERTY FieldOfView : REFERENCE TO FieldOfView
GET
END_GET
END_PROPERTY

END_INTERFACE

// ---- Context/MainStation.TcPOU
FUNCTION_BLOCK MainStation EXTENDS TcoCore.TcoObject
//VAR
//    turckRfidHead : RfidHead(THIS^, T#1MS);
//    sUId          : T_MaxString;
//END_VAR
//VAR
//	    _uid          : BOOL;
//END_VAR

VAR
    //    rfidHead_Test : IVController_Test;

END_VAR

//TcUnit.RUN();

END_FUNCTION_BLOCK

// ---- Context/PRG_TEST.TcPOU
PROGRAM PRG_TEST
VAR
    _testSuite : TcUnitContext;
END_VAR

_testSuite.Run();
_testSuite.RtcSynchronize(true, '', 60);

END_PROGRAM

// ---- Context/TcUnitContext.TcPOU
FUNCTION_BLOCK TcUnitContext EXTENDS TcoCore.TcoContext
VAR
    _mainStation : MainStation(THIS^);

    {attribute addProperty Name "Versionsnummer Plc"}
    _sVersion : STRING(23);
    //~
    _stProgramVersion : ST_LibVersion;
    //~

END_VAR

(*~
    <docu>
        <summary>
            Main method of the TcoContext. This is the entry point of any control logic that belongs to this context.
            The call of this method is ensured by calling the <c>InstanceName.Run()</c> method, and it must not be called explicitly.
            This method is abstract, and it must be overridden in derived block.
        </summary>
    </docu>
~*)
METHOD PROTECTED Main

_mainStation();
END_METHOD

END_FUNCTION_BLOCK

// ---- IV3/IVController.TcPOU
FUNCTION_BLOCK IVController EXTENDS TcoCore.TcoComponent
VAR
    _triggerSensorTask        : TriggerSensor(THIS^);
    _readTool1CoordinatesTask : ReadCoordinates(THIS^, CoeIndex := Tool1CoeIndex);
    _readTool2CoordinatesTask : ReadCoordinates(THIS^, CoeIndex := Tool2CoeIndex);
    _readTool3CoordinatesTask : ReadCoordinates(THIS^, CoeIndex := Tool3CoeIndex);

    _calculationTask : CalculationTask
    (
        THIS^
        , ResolutionX := 1280
        , ResolutionY := 960
        , OffsetY     := -7.0129
        , GainY       := 2.5438
        , OffsetX     := -5.57888
        , GainX       := 3.387877
    );
END_VAR

VAR
    _fb_coe_write       : FB_EcCoESdoWrite; // Function Block for writing in CoE
    _fb_coe_read        : FB_EcCoESdoRead;  // Function Block for reading from CoE
    userNetId           : T_AmsNetId;       // Have to be entered
    _startWrite         : BOOL := FALSE;    // Sign for start writing
    _startRead          : BOOL := FALSE;    // Sign for start reading
    _nState             : BYTE := 0;        // RW-status
    _int16Buffer        : INT;              // Buffer for reading
    _uint16Buffer       : UINT := 22;       // Buffer for writing
    _bTxPDOState AT %I* : BOOL;             // (PDO for synchronization)
    AdsErrId            : UDINT;
    CANopenErrId        : UDINT;

    _index             : UINT := 16#1008;
    _subIndex          : BYTE := 0;
    _result            : STRING;
    _stringBuffer      : STRING;
    _numberBuffer      : UDINT;
    _exe               : BOOL;
    _generalDeviceInfo : GeneralDeviceInformation;
    _IdentityCoe       : IdentityCoe;
    _coordinates       : Coordinates;
    _readCoordinates   : BOOL;
END_VAR
VAR CONSTANT
    Tool1CoeIndex : UINT := 16#8015;
    Tool2CoeIndex : UINT := 16#8025;
    Tool3CoeIndex : UINT := 16#8035;

END_VAR
VAR

    //    //Ethercat Status
    //~
    StatusOfSystem AT %I* : Status_of_System;
    //PDO Vision Sensor   
    InputResponse                                 AT %I* : Input_Response;
    ID01_CurrentValue                             AT %I* : ID01_Current_Value;
    ID02_MatchingRateOfPositionAdujustmentTool_01 AT %I* : ID02_Current_Value; //value 0..1
    ID03_MatchingRateOfPositionAdujustmentTool_02 AT %I* : ID03_Current_Value; //value 0..1
    ID04_MatchingRateOfPositionAdujustmentTool_03 AT %I* : ID04_Current_Value; //value 0..1
    ID05_MatchingRateOfPositionAdujustmentTool_04 AT %I* : ID05_Current_Value; //value 0..1
    ID06_MatchingRateOfPositionAdujustmentTool_05 AT %I* : ID06_Current_Value; //value 0..1
    ID07_MatchingRateOfPositionAdujustmentTool_06 AT %I* : ID07_Current_Value; //value 0..1
    ID08_MatchingRateOfPositionAdujustmentTool_07 AT %I* : ID08_Current_Value; //value 0..1
    ID01Status                                    AT %I* : ID01_Status;
    _ID01Status                                          : ID01_Status := ID01Status;

    ID02Status   AT %I* : ID02_Status;
    ID03Status   AT %I* : ID03_Status;
    ID04Status   AT %I* : ID04_Status;
    ID05Status   AT %I* : ID05_Status;
    ID06Status   AT %I* : ID06_Status;
    ID07Status   AT %I* : ID07_Status;
    ID08Status   AT %I* : ID08_Status;
    InputRequest AT %Q* : Input_Request;
    //    //General Ethercat Data
    WcState  AT %I* : WcState_0B2B16F9;
    InfoData AT %I* : InfoData;
    //~

    _trigger        : BOOL;
    _readString     : BOOL;
    _readDeviceInfo : BOOL;
END_VAR

////////////////////////////////////////////
_triggerSensorTask
(
    Iv3InputRequest1    := THIS^.InputRequest.Request_1
    , Iv3InputResponse1 := THIS^.InputResponse.Response_1
    , StatusOfSystem    := THIS^.StatusOfSystem
    , ActionDesc        := '<#TriggerSensor#>'
);

_readTool1CoordinatesTask
(
    InfoData         := THIS^.InfoData
    , StatusOfSystem := THIS^.StatusOfSystem
    , ResultValue    := THIS^.ID02_MatchingRateOfPositionAdujustmentTool_01.Tool_00_Score
    , ActionDesc     := '<#ReadCoordinates Tool1#>'
);

_readTool2CoordinatesTask
(
    InfoData         := THIS^.InfoData
    , StatusOfSystem := THIS^.StatusOfSystem
    , ResultValue    := THIS^.ID03_MatchingRateOfPositionAdujustmentTool_02.Tool_01_Score
    , ActionDesc     := '<#ReadCoordinates Tool2#>'
);

_readTool3CoordinatesTask
(
    InfoData         := THIS^.InfoData
    , StatusOfSystem := THIS^.StatusOfSystem
    , ResultValue    := THIS^.ID04_MatchingRateOfPositionAdujustmentTool_03.Tool_02_Score
    , ActionDesc     := '<#ReadCoordinates Tool3#>'
);

_calculationTask
(
    InfoData           := THIS^.InfoData
    , StatusOfSystem   := THIS^.StatusOfSystem
    , CoordinatesTool1 := _readTool1CoordinatesTask.RawCoordinates
    , CoordinatesTool2 := _readTool2CoordinatesTask.RawCoordinates
    , CoordinatesTool3 := _readTool3CoordinatesTask.RawCoordinates
    , ActionDesc       := '<#_calculationTask#>'
);

/////////////////////////////////////////////
//IF _trigger THEN
//    THIS^.InputRequest.Request_1.Trigger := TRUE;

//    IF THIS^.InputResponse.Response_1.Trigger THEN
//        _trigger                             := FALSE;
//        THIS^.InputRequest.Request_1.Trigger := FALSE;
//    end_if
//END_IF

userNetId := Tc2_System.F_CreateAmsNetId(THIS^.InfoData.AdsAddr.netId);

IF _readString THEN
    _stringBuffer := CoeReadString(_index := _index, _subIndex := _subIndex);
END_IF

IF _readDeviceInfo THEN

    IF GeneralDeviceInfo() THEN
        _readDeviceInfo := false;
    END_IF
END_IF

CoeReadIdentity();

IF _readCoordinates THEN
    IF CoeReadCoordinates() THEN
        _readCoordinates := FALSE;
    END_IF

END_IF

_ID01Status := ID01Status;

METHOD CalculationMethod : TcoCore.ITcoTaskStatus
IF (CalculationTask <> 0) THEN
    CalculationMethod := CalculationTask.Invoke();
END_IF
END_METHOD

PROPERTY CalculationTask : iCalculationTask
GET
CalculationTask := _calculationTask;
END_GET
END_PROPERTY

METHOD CoeReadCoordinates : BOOL
VAR_INST
    step : UINT := 1;

END_VAR
CASE step OF
    1:
        CoeReadCoordinates := FALSE;
        step               := 10;
    10:
        _coordinates.xValue := CoeReadUDINT
        (
            _index      := 16#8015
            , _subIndex := 16#11
        );

        IF NOT _fb_coe_read.bBusy THEN
            step := 20;
        END_IF
    20:
        _coordinates.yValue := CoeReadUDINT
        (
            _index      := 16#8015
            , _subIndex := 16#12
        );

        IF NOT _fb_coe_read.bBusy THEN
            step := 40;
        END_IF
    40:
        _coordinates.variableValue := CoeReadUDINT
        (
            _index      := 16#8015
            , _subIndex := 16#13
        );

        IF NOT _fb_coe_read.bBusy THEN
            step               := 1;
            CoeReadCoordinates := TRUE;
        END_IF
END_CASE
END_METHOD

METHOD CoeReadIdentity : UDINT
VAR_INST
    _fb_coe_read_ext   : Tc2_EtherCAT.FB_EcCoESdoReadEx;
    _timeout           : TIME := DEFAULT_ADS_TIMEOUT;
    _identityCoeToSwap : IdentityCoe;

    i     : UINT;
    _test : STRING;
END_VAR

// Read entry
_fb_coe_read_ext
(
    sNetId            := userNetId
    , nSlaveAddr      := InfoData.AdsAddr.port
    , nSubIndex       := 0
    , nIndex          := 16#1018
    , pDstBuf         := ADR(_identityCoeToSwap)
    , cbBufLen        := 32
    , bExecute        := true
    , tTimeout        := _timeout
    , bCompleteAccess := TRUE
);

IF _fb_coe_read.bError THEN
    _nState := 100; // Error case
ELSE

    IF NOT _fb_coe_read.bBusy THEN
        _IdentityCoe.ProductKey   := SHR(_identityCoeToSwap.ProductKey, 16);
        _IdentityCoe.VendorId     := SHR(_identityCoeToSwap.VendorId, 16);
        _IdentityCoe.Revision     := SHR(_identityCoeToSwap.Revision, 16);
        _IdentityCoe.SerialNumber := SHR(_identityCoeToSwap.SerialNumber, 16);
        _fb_coe_read(bExecute := FALSE);
        _readString := false;
    END_IF

END_IF
END_METHOD

METHOD CoeReadString : STRING
//VAR_INST
//    _stringBuffer : STRING;
//END_VAR
VAR_INPUT
    _index    : UINT;
    _subIndex : BYTE;
END_VAR

// Read entry
_fb_coe_read
(
    sNetId       := userNetId
    , nSlaveAddr := InfoData.AdsAddr.port
    //    , nSlaveAddr := 1001
    , nSubIndex := _subIndex
    , nIndex    := _index
    , pDstBuf   := ADR(_stringBuffer)
    , cbBufLen  := 12
    , bExecute  := true
    , tTimeout  := T#1S
);

IF _fb_coe_read.bError THEN
    AdsErrId := _fb_coe_read.nErrId;
ELSE
    IF NOT _fb_coe_read.bBusy THEN
        _fb_coe_read(bExecute := FALSE);
        _readString := false;
    END_IF
END_IF

CoeReadString := _stringBuffer;
END_METHOD

METHOD CoeReadUDINT : UDINT
//VAR_INST
//    _stringBuffer : STRING;
//END_VAR
VAR_INPUT
    _index    : UINT;
    _subIndex : BYTE;
END_VAR

// Read entry
_fb_coe_read
(
    sNetId       := userNetId
    , nSlaveAddr := InfoData.AdsAddr.port
    //    , nSlaveAddr := 1001
    , nSubIndex := _subIndex
    , nIndex    := _index
    , pDstBuf   := ADR(_numberBuffer)
    , cbBufLen  := 32
    , bExecute  := true
    , tTimeout  := T#1S
);

IF _fb_coe_read.bError THEN
    _nState := 100; // Error case
ELSE
    IF NOT _fb_coe_read.bBusy THEN
        _fb_coe_read(bExecute := FALSE);
        _readString := false;
    END_IF
END_IF

CoeReadUDINT := _numberBuffer;
END_METHOD

{attribute 'monitoring' := 'call'}
PROPERTY ErrorId : UINT
GET
ErrorId := THIS^.StatusOfSystem.Error_Code or _readTool1CoordinatesTask.ErrorId or _triggerSensorTask.ErrorId;
END_GET
END_PROPERTY

METHOD PRIVATE GeneralDeviceInfo : BOOL;
VAR_INST
    step : UINT := 1;

END_VAR
CASE step OF
    1:
        GeneralDeviceInfo := FALSE;
        step              := 10;
    10:
        _generalDeviceInfo.DeviceName := CoeReadString
        (
            _index      := 16#1008
            , _subIndex := 0
        );

        IF NOT _fb_coe_read.bBusy THEN
            step := 20;
        END_IF
    20:
        step := 25;
    25:
        _generalDeviceInfo.HardwareVersion := CoeReadString
        (
            _index      := 16#1009
            , _subIndex := 0
        );

        IF NOT _fb_coe_read.bBusy THEN
            step := 30;
        END_IF
    30:
        step := 35;
    35:
        _generalDeviceInfo.DeviceType := CoeReadUDINT
        (
            _index      := 16#1000
            , _subIndex := 0
        );

        IF NOT _fb_coe_read.bBusy THEN
            step := 40;
        END_IF
    40:
        GeneralDeviceInfo := FALSE;
        step              := 45;
    45:
        _generalDeviceInfo.SoftwareVersion := CoeReadString
        (
            _index      := 16#100A
            , _subIndex := 0
        );

        IF NOT _fb_coe_read.bBusy THEN
            step              := 1;
            GeneralDeviceInfo := TRUE;
        END_IF

END_CASE
END_METHOD

{attribute 'monitoring' := 'call'}
PROPERTY ID01StatusProp : REFERENCE TO ID01_Status
GET
ID01StatusProp REF= _ID01Status;
END_GET
END_PROPERTY

{attribute 'monitoring' := 'call'}
PROPERTY IsError : BOOL
GET
//collected Error from Tasks
IsError := statusOfSystem.Error_Status OR TriggerSensorTask.Error or ReadTool1CoordinatesTask.Error;
END_GET
END_PROPERTY

PROPERTY RawCoordinatesTool1 : REFERENCE TO Coordinates
GET
RawCoordinatesTool1 REF= _readTool1CoordinatesTask.RawCoordinates;
END_GET
END_PROPERTY

PROPERTY RawCoordinatesTool2 : REFERENCE TO Coordinates
GET
RawCoordinatesTool2 REF= _readTool2CoordinatesTask.RawCoordinates;
END_GET
END_PROPERTY

PROPERTY RawCoordinatesTool3 : REFERENCE TO Coordinates
GET
RawCoordinatesTool3 REF= _readTool3CoordinatesTask.RawCoordinates;
END_GET
END_PROPERTY

METHOD ReadTool1CoordinatesMethod : TcoCore.ITcoTaskStatus
IF (ReadTool1CoordinatesTask <> 0) THEN
    ReadTool1CoordinatesMethod := ReadTool1CoordinatesTask.Invoke();
END_IF
END_METHOD

PROPERTY ReadTool1CoordinatesTask : TcoCore.ITcoTask
GET
ReadTool1CoordinatesTask := _readTool1CoordinatesTask;
END_GET
END_PROPERTY

METHOD ReadTool2CoordinatesMethod : TcoCore.ITcoTaskStatus
IF (ReadTool2CoordinatesTask <> 0) THEN
    ReadTool2CoordinatesMethod := ReadTool2CoordinatesTask.Invoke();
END_IF
END_METHOD

PROPERTY ReadTool2CoordinatesTask : TcoCore.ITcoTask
GET
ReadTool2CoordinatesTask := _readTool2CoordinatesTask;
END_GET
END_PROPERTY

METHOD ReadTool3CoordinatesMethod : TcoCore.ITcoTaskStatus
IF (ReadTool3CoordinatesTask <> 0) THEN
    ReadTool3CoordinatesMethod := ReadTool3CoordinatesTask.Invoke();
END_IF
END_METHOD

PROPERTY ReadTool3CoordinatesTask : TcoCore.ITcoTask
GET
ReadTool3CoordinatesTask := _readTool3CoordinatesTask;
END_GET
END_PROPERTY

(*~
    <docu>
        <summary>
            Restore all tasks of this instance into initial state.
        </summary>
    </docu>
~*)
METHOD Restore : ITcoRestorable

IF (TriggerSensorTask <> 0) THEN
    TriggerSensorTask.Restore();
END_IF;

IF (ReadTool1CoordinatesTask <> 0) THEN
    ReadTool1CoordinatesTask.Restore();
END_IF;

//IF (WriteDataTask) <> 0 THEN
//    WriteDataTask.Restore();
//END_IF

//IF (LockTask) <> 0 THEN
//    LockTask.Restore();
//END_IF

//IF (ResetTask) <> 0 THEN
//    ResetTask.Restore();
//END_IF
END_METHOD

PROPERTY ScoreToolHeight : DINT
GET
ScoreToolHeight := ID03_MatchingRateOfPositionAdujustmentTool_02.Tool_01_Score;
END_GET
END_PROPERTY

PROPERTY ScoreToolPositionCorrector : DINT
GET
ScoreToolPositionCorrector := ID02_MatchingRateOfPositionAdujustmentTool_01.Tool_00_Score;
END_GET
END_PROPERTY

PROPERTY ScoreToolWidth : DINT
GET
ScoreToolWidth := ID04_MatchingRateOfPositionAdujustmentTool_03.Tool_02_Score;
END_GET
END_PROPERTY

METHOD PROTECTED ServiceMode
END_METHOD

METHOD TriggerSensorMethod : TcoCore.ITcoTaskStatus
IF (TriggerSensorTask <> 0) THEN
    TriggerSensorMethod := TriggerSensorTask.Invoke();
END_IF
END_METHOD

PROPERTY TriggerSensorTask : TcoCore.ITcoTask
GET
TriggerSensorTask := _triggerSensorTask;
END_GET
END_PROPERTY

END_FUNCTION_BLOCK

// ---- IV3/Tasks/TriggerSensor.TcPOU
FUNCTION_BLOCK TriggerSensor EXTENDS TcoCore.TcoTask
VAR_IN_OUT
    Iv3InputRequest1  : Iv3InputRequestResponse1;
    Iv3InputResponse1 : Iv3InputRequestResponse1;
    StatusOfSystem    : Status_of_System;
END_VAR
VAR_INPUT
    ActionDesc : STRING(25);
END_VAR
VAR
    _state   : USINT;
    _errorId : UINT;

END_VAR

IF (THIS^.Execute()) THEN
    //ERror Case
    THIS^.ThrowWhen(StatusOfSystem.Error_Status);

    CASE _state OF
        10:
            Iv3InputRequest1.Trigger := TRUE;
            _state                   := 20;
        20:
            THIS^.DoneWhen(Iv3InputResponse1.Trigger);
    END_CASE
END_IF

{attribute 'monitoring' := 'call'}
PROPERTY ErrorId : UINT
GET
ErrorId := _errorId;
END_GET
END_PROPERTY

METHOD PUBLIC FB_init : BOOL
VAR_INPUT
    bInitRetains : BOOL; // if TRUE, the retain variables are initialized (warm start / cold start)
    bInCopyCode  : BOOL; // if TRUE, the instance afterwards gets moved into the copy code (online change)
    ParentObject : ITcoObject;
END_VAR
// This is not clear to me... I from time to time the consumer code does not see 'FB_init' of 'TcoObject', that's why overridden here with super call...
{warning disable C0316}
SUPER^.FB_init(bInitRetains, bInCopyCode, ParentObject);
END_METHOD

(*~
    <docu>
        <summary>
            Executes when task reaches the ```Done``` state .
        </summary>
    </docu>
~*)
METHOD PROTECTED OnDone
{warning disable C0371}
Iv3InputRequest1.Trigger := FALSE;
//this^.Restore();
END_METHOD

(*~
    <docu>
        <summary>
            Executes when task reaches the ```Error``` state.
            <para>
                Do not confuse with <see cref="PlcDocu.TcoCore.TcoTask.WhileError()"/>, that is called cyclically until '''Error''' state is left.
            </para>
        </summary>
    </docu>
~*)
METHOD PROTECTED OnError
{warning disable C0371}
_errorId := StatusOfSystem.Error_Code;
END_METHOD

(*~
	<docu>
		<summary>
			Executes ones when the task starts (at the moment of transition from the ```Requested``` state into the ```Busy``` state).
		</summary>			
	</docu>	
~*)
METHOD PROTECTED OnStart
{warning disable C0371}
_state := 10;
END_METHOD

(*~
    <docu>
        <summary>
            Restores this instance to the Ready state. Can be called explicitly or from within one of the restore mechanisms.
            <para>
                See also <see cref="PlcDocu.TcoCore.TcoTask.AutoRestorable()"/>
            </para>
        </summary>
    </docu>
~*)
METHOD Restore : ITcoRestorable
{warning disable C0371}
Iv3InputRequest1.Trigger    := FALSE;
Iv3InputRequest1.ResetError := TRUE;

IF Iv3InputResponse1.ResetError THEN
    Iv3InputRequest1.ResetError := FALSE;
END_IF
END_METHOD

END_FUNCTION_BLOCK

// ---- IV3/Tasks/ReadCoordinates.TcPOU
FUNCTION_BLOCK ReadCoordinates EXTENDS TcoCore.TcoTask
VAR_IN_OUT
    InfoData       : InfoData;
    StatusOfSystem : Status_of_System;
    ResultValue    : DINT;
END_VAR
VAR_INPUT
    ActionDesc : STRING(25);
END_VAR
VAR
    _fb_coe_read_ext : Tc2_EtherCAT.FB_EcCoESdoReadEx;
    _timeout         : TIME := Tc2_System.DEFAULT_ADS_TIMEOUT;
    _state           : INT  := 10;
    _data            : ARRAY[1..31] OF DINT;
    _errorId         : UDINT;
    _rawCoordinates  : Coordinates;
    _coeIndex        : UINT;

END_VAR
VAR CONSTANT
    SIZE_OF_TWO_BYTES : UINT := 16;
END_VAR

IF (THIS^.Execute()) THEN
    //ERror Case

    THIS^.ThrowWhen(StatusOfSystem.Error_Status);

    CASE _state OF
        10:
            _fb_coe_read_ext
            (
                sNetId            := Tc2_System.F_CreateAmsNetId(infodata.AdsAddr.netId)
                , nSlaveAddr      := InfoData.AdsAddr.port
                , nSubIndex       := 16#0
                , nIndex          := _coeIndex
                , pDstBuf         := ADR(_data)
                , cbBufLen        := SIZEOF(_data) + 2
                , tTimeout        := _timeout
                , bCompleteAccess := TRUE
            );

            _state := 20;
        20:
            _fb_coe_read_ext(bExecute := TRUE);
            _state := 30;
        30:
            _fb_coe_read_ext();

            IF _fb_coe_read_ext.bBusy THEN
                RETURN;
            END_IF

            IF _fb_coe_read_ext.bError THEN
                _State := 99; // Error case
                RETURN;
            END_IF

            _rawCoordinates.xValue        := SHR(_data[017], SIZE_OF_TWO_BYTES);
            _rawCoordinates.yValue        := SHR(_data[018], SIZE_OF_TWO_BYTES);
            _rawCoordinates.variableValue := SHR(_data[019], SIZE_OF_TWO_BYTES);

            _state := 80;
        40:
            //            Calculating
            //            (
            //                ResolutionY := ReadCoordinates.ResolutionY
            //                , PixelY    := _rawCoordinates.variableValue
            //                , ValueY    := THIS^.ResultValue
            //                , ResolutionX := ReadCoordinates.ResolutionX
            //                , PixelX := _rawCoordinates.
            //                , ValueX
            //                , FieldOfView => _fieldOfView
            //                , Distance    => _distanceFromHeight
            //            );

            _state := 80;

        50: // Calculate the Position in mm with FOV and Distance

        80:

            THIS^.DoneWhen(TRUE);
        99:
            THIS^.ThrowWhen(TRUE);

    END_CASE
END_IF

{attribute 'monitoring' := 'call'}
PROPERTY ErrorId : UINT
GET
ErrorId := udint_to_uint(_errorId);
END_GET
END_PROPERTY

METHOD PUBLIC FB_init : BOOL
VAR_INPUT
    bInitRetains : BOOL; // if TRUE, the retain variables are initialized (warm start / cold start)
    bInCopyCode  : BOOL; // if TRUE, the instance afterwards gets moved into the copy code (online change)
    ParentObject : ITcoObject;
    CoeIndex     : UINT;
END_VAR
// This is not clear to me... I from time to time the consumer code does not see 'FB_init' of 'TcoObject', that's why overridden here with super call...
{warning disable C0316}
SUPER^.FB_init(bInitRetains, bInCopyCode, ParentObject);

_coeIndex := CoeIndex;
END_METHOD

(*~
    <docu>
        <summary>
            Executes when task reaches the ```Done``` state .
        </summary>
    </docu>
~*)
METHOD PROTECTED OnDone
{warning disable C0371}
_fb_coe_read_ext(bExecute := False);
END_METHOD

(*~
    <docu>
        <summary>
            Executes when task reaches the ```Error``` state.
            <para>
                Do not confuse with <see cref="PlcDocu.TcoCore.TcoTask.WhileError()"/>, that is called cyclically until '''Error''' state is left.
            </para>
        </summary>
    </docu>
~*)
METHOD PROTECTED OnError
{warning disable C0371}
_fb_coe_read_ext(nErrId => _errorId);
END_METHOD

(*~
	<docu>
		<summary>
			Executes ones when the task starts (at the moment of transition from the ```Requested``` state into the ```Busy``` state).
		</summary>			
	</docu>	
~*)
METHOD PROTECTED OnStart
{warning disable C0371}
_fb_coe_read_ext(bExecute := FALSE);
_state := 10;
END_METHOD

PROPERTY RawCoordinates : REFERENCE TO Coordinates
GET
RawCoordinates REF= _rawCoordinates;
END_GET
END_PROPERTY

(*~
    <docu>
        <summary>
            Restores this instance to the Ready state. Can be called explicitly or from within one of the restore mechanisms.
            <para>
                See also <see cref="PlcDocu.TcoCore.TcoTask.AutoRestorable()"/>
            </para>
        </summary>
    </docu>
~*)
METHOD Restore : ITcoRestorable
{warning disable C0371}
_fb_coe_read_ext(bExecute := FALSE);
END_METHOD

END_FUNCTION_BLOCK

// ---- IV3/Tasks/CalculationTask.TcPOU
FUNCTION_BLOCK CalculationTask EXTENDS TcoCore.TcoTask IMPLEMENTS iCalculationTask
VAR_IN_OUT
    InfoData         : InfoData;
    StatusOfSystem   : Status_of_System;
    CoordinatesTool1 : Coordinates;
    CoordinatesTool2 : Coordinates;
    CoordinatesTool3 : Coordinates;
END_VAR
VAR_INPUT
    ActionDesc : STRING(25);
END_VAR
VAR
    _data                    : ARRAY[1..31] OF DINT;
    _errorId                 : UDINT;
    _coeIndex                : UINT;
    _distanceFromX           : LREAL;
    _distanceFromY           : LREAL;
    _fieldOfView             : FieldOfView;
    _coordinatesInMillimeter : Coordinates;

    _resolutionX : UINT;
    _resolutionY : UINT;

    _states : (CalculatingCoefficientState
        , CalculatingFieldOfViewState
        , CalculatingDistanceState
        , CaulculatingCoordinatesInMillimeter
        , DoneState
        , ErrorState);

    //lineare Regression
    _offsetX      : LREAL;
    _gainX        : LREAL;
    _coefficientX : LREAL;

    _offsetY      : LREAL;
    _gainY        : LREAL;
    _coefficientY : LREAL;
END_VAR
//in mm     Breite			
//50		16,4		   22,4 
//100		31,2		   42,1 
//200		60,7		   81,4 
//300		90,2		   120,7
//400		119,7		   160,0
//500		149,2		   199,3
//600		178,7		   238,6
//700		208,3		   277,9
//800		237,8		   317,2
//900		267,3		   356,6
//1000		296,8	       395,9
//1250		370,6	       494,2
//1500		444,4	       592,4
//1750		518,2	       690,7
//2000		592		       789

IF (THIS^.Execute()) THEN
    //ERror Case

    THIS^.ThrowWhen(StatusOfSystem.Error_Status);

    CASE _states OF
        CalculatingCoefficientState:
            _coefficientX := CalcCoefficientFromResolutionAndPixel
            (
                Resolution := _resolutionX
                , Pixel    := CoordinatesTool3.variableValue
            );

            _coefficientY := CalcCoefficientFromResolutionAndPixel
            (
                Resolution := _resolutionY
                , Pixel    := CoordinatesTool2.variableValue
            );

            _states := CalculatingFieldOfViewState;

        CalculatingFieldOfViewState:

            FieldOfView.xValue :=
                CalcFieldOfViewWithCoefficientAndObjectMeasurement
            (
                Coefficient := _coefficientX
                , Value     := THIS^.ControllerRef.ScoreToolWidth
            );

            FieldOfView.yValue :=
                CalcFieldOfViewWithCoefficientAndObjectMeasurement
            (
                Coefficient := _coefficientY
                , Value     := THIS^.ControllerRef.ScoreToolHeight
            );

            _states := CalculatingDistanceState;

        CalculatingDistanceState:

            _distanceFromX := (FieldOfView.xValue * _gainX) + _offsetX;
            _distanceFromY := (FieldOfView.yValue * _gainY) + _offsetY;
            _states        := CaulculatingCoordinatesInMillimeter;

        CaulculatingCoordinatesInMillimeter:
            _coordinatesInMillimeter.xValue :=
                LREAL_TO_DINT((FieldOfView.xValue / _resolutionX) * CoordinatesTool1.xValue);

            _coordinatesInMillimeter.yValue :=
                LREAL_TO_DINT((FieldOfView.yValue / _resolutiony) * CoordinatesTool1.yValue);

            _coordinatesInMillimeter.variableValue := CoordinatesTool1.variableValue;

            _states := DoneState;

        DoneState:

            THIS^.DoneWhen(TRUE);
        ErrorState:
            THIS^.ThrowWhen(TRUE);

    END_CASE
END_IF

METHOD PROTECTED CalcCoefficientFromResolutionAndPixel : LREAL
VAR_INPUT
    Resolution : LREAL;
    Pixel      : LREAL;
END_VAR

IF Pixel = 0 THEN
    THIS^.Messenger.Error('Was ist los mit dir, teile nicht durch 0!');
    CalcCoefficientFromResolutionAndPixel := 0;
    RETURN;
END_IF

CalcCoefficientFromResolutionAndPixel := (Resolution / Pixel) * 10;
END_METHOD

METHOD PRIVATE CalcFieldOfViewWithCoefficientAndObjectMeasurement : LREAL
VAR_INPUT
    Coefficient : LREAL;
    Value       : DINT;
END_VAR
CalcFieldOfViewWithCoefficientAndObjectMeasurement := (Coefficient * DWORD_TO_LREAL(Value)) / 100;
END_METHOD

PROPERTY ControllerRef : REFERENCE TO IVController
GET
VAR
    _controllerRef : POINTER TO IVController;
END_VAR
IF __QUERYPOINTER(_ParentObject, _controllerRef) THEN // Check if _Parent is Station001
    ControllerRef REF= _controllerRef^;               // If the check is successful dereference a pointer. simlar to THIS^ or SUPER^
END_IF
END_GET
END_PROPERTY

PROPERTY CoordinatesInMillimeter : REFERENCE TO Coordinates
GET
CoordinatesInMillimeter Ref= _coordinatesInMillimeter;
END_GET
END_PROPERTY

PROPERTY DistanceFromObject : LREAL
GET
IF (_distanceFromX <> 0 AND _distanceFromY <> 0) THEN
    DistanceFromObject := (_distanceFromX + _distanceFromY) / 2;
ELSE
    DistanceFromObject := 0;
END_IF
END_GET
END_PROPERTY

{attribute 'monitoring' := 'call'}
PROPERTY ErrorId : UINT
GET
ErrorId := udint_to_uint(_errorId);
END_GET
END_PROPERTY

METHOD PUBLIC FB_init : BOOL
VAR_INPUT
    bInitRetains : BOOL; // if TRUE, the retain variables are initialized (warm start / cold start)
    bInCopyCode  : BOOL; // if TRUE, the instance afterwards gets moved into the copy code (online change)
    ParentObject : ITcoObject;
    ResolutionX  : UINT;
    ResolutionY  : UINT;
    OffsetX      : LREAL;
    GainX        : LREAL;
    OffsetY      : LREAL;
    GainY        : LREAL;

END_VAR
// This is not clear to me... I from time to time the consumer code does not see 'FB_init' of 'TcoObject', that's why overridden here with super call...
{warning disable C0316}
SUPER^.FB_init(bInitRetains, bInCopyCode, ParentObject);

THIS^._resolutionX := ResolutionX;
THIS^._resolutionY := ResolutionY;

_offsetX := OffsetX;
_gainX   := GainX;
_offsetY := OffsetY;
_gainY   := GainY;
END_METHOD

PROPERTY FieldOfView : REFERENCE TO FieldOfView
GET
FieldOfView REF= _fieldOfView;
END_GET
END_PROPERTY

(*~
    <docu>
        <summary>
            Executes when task reaches the ```Done``` state .
        </summary>
    </docu>
~*)
METHOD PROTECTED OnDone
{warning disable C0371}
//this^.Restore();
END_METHOD

(*~
    <docu>
        <summary>
            Executes when task reaches the ```Error``` state.
            <para>
                Do not confuse with <see cref="PlcDocu.TcoCore.TcoTask.WhileError()"/>, that is called cyclically until '''Error''' state is left.
            </para>
        </summary>
    </docu>
~*)
METHOD PROTECTED OnError
{warning disable C0371}
END_METHOD

(*~
	<docu>
		<summary>
			Executes ones when the task starts (at the moment of transition from the ```Requested``` state into the ```Busy``` state).
		</summary>			
	</docu>	
~*)
METHOD PROTECTED OnStart
{warning disable C0371}
_states := CalculatingCoefficientState;
END_METHOD

(*~
    <docu>
        <summary>
            Restores this instance to the Ready state. Can be called explicitly or from within one of the restore mechanisms.
            <para>
                See also <see cref="PlcDocu.TcoCore.TcoTask.AutoRestorable()"/>
            </para>
        </summary>
    </docu>
~*)
METHOD Restore : ITcoRestorable
{warning disable C0371}
END_METHOD

END_FUNCTION_BLOCK

// ---- Project Information/F_GetCompany.TcPOU
// This function has been automatically generated from the project information.
{attribute 'signature_flag' := '1073741824'}
{attribute 'TcGenerated'}
{attribute 'no-analysis'}
FUNCTION F_GetCompany : WSTRING
VAR_INPUT

END_VAR

F_GetCompany := "Gema";

END_FUNCTION

// ---- Project Information/F_GetTitle.TcPOU
// This function has been automatically generated from the project information.
{attribute 'signature_flag' := '1073741824'}
{attribute 'TcGenerated'}
{attribute 'no-analysis'}
FUNCTION F_GetTitle : WSTRING
VAR_INPUT

END_VAR

F_GetTitle := "LibraryVision";

END_FUNCTION

// ---- Project Information/F_GetVersion.TcPOU
// This function has been automatically generated from the project information.
{attribute 'signature_flag' := '1073741824'}
{attribute 'TcGenerated'}
{attribute 'no-analysis'}
FUNCTION F_GetVersion : ST_LibVersion
VAR_INPUT

END_VAR

F_GetVersion.iMajor    := 0;
F_GetVersion.iMinor    := 9;
F_GetVersion.iBuild    := 9;
F_GetVersion.iRevision := 9;
F_GetVersion.sVersion  := '0.9.9.9';
F_GetVersion.nFlags    := 0;

END_FUNCTION
